Staubli VAL3: onF1Event.pgx

program onF1Event()
  local bool l_bLoop
begin
  // look if the bButton is enable
  if bButton[0]
    //
    //  Set the LOOP ON/OFF
    //
    logMsg("[KERNEL] INTERFACE:Change the loop status")
    call processList:getLoop(l_bLoop)
    call processList:setLoop(!l_bLoop)
  endIf
end
